(* Logix 5000 project; controller cal1615 1756-L62 rev 20.19; software revision 20.05; part 26 of 82 *)
(* tags used below, declared in another part *)
   AFI : BOOL;   // Always False Bit
   FAULT : BOOL;   // Fault AFI
   p01_param_open_oven_temp : REAL;
   p01_recipe_active : recipe;   // Active Recipe
   p01_sys_enc : SYS_ENC;   // System Encoder
   p01r09_open_oven : BOOL;
   p01r09_pb_global_reset : BOOL;   // System Modes PB: Global Fault Reset
   p01r13_permissive_oxidizer : BOOL;   // System Line Start Sequence Permissive Oxidizer
   p02_dint_from_hmi : hmi_dint;
   p11r30 : routine;   // Zone 1 Temperature Control
   p12_ai_lfl : REAL;   // Zone 2 Analog Input Lower Flash Limit
   p12_ai_tc01 : REAL;   // Zone 2 Analog Input Control Thermocouple 1
   p12_ai_tc02 : REAL;   // Zone 2 Analog Input Control Thermocouple 2
   p12_ao_cv : REAL;   // Zone 2 Analog Output Control Valve
   p12_di_burner_auto : BOOL;   // Zone 2 Digital Input Burner Auto
   p12_di_burner_safeties_ok : BOOL;   // Zone 2 Digital Input Burner Safeties Ok
   p12_di_door_open : BOOL;   // Zone 2 Digital Input Access Door Open
   p12_di_exh : acs800_di_normal;   // Zone 2 Digital Inputs Exhaust Fan
   p12_di_exh_flow_ok : BOOL;   // Zone 2 Digital Input Exhaust Flow OK
   p12_di_flame_failure : BOOL;   // Zone 2 Digital Input Flame Failure
   p12_di_flame_on : BOOL;   // Zone 2 Digital Input Burner is On
   p12_di_high_limit_temp_ok : BOOL;   // Zone 2 Digital Input High Limit Temperature OK
   p12_di_recirc : acs800_di_normal;   // Zone 2 Digital Inputs Recirc Fan
   p12_di_recirc_flow_ok : BOOL;   // Zone 2 Digital Input Recirc Flow OK
   p12_di_sp00 : BOOL;   // Zone 2 Digital Input Combustion Blower Pressure OK
   p12_di_tc01_bo : BOOL;   // Zone 2 Digital Input Control Thermocouple 1 Failure
   p12_di_tc02_bo : BOOL;   // Zone 2 Digital Input Control Thermocouple 2 Failure
   p12_do_enable_burner : BOOL;   // Zone 2 Digital Output Enable Burner
   p12_do_rst_flame : BOOL;   // Zone 2 Digital Output Reset Flame Safety
   p12_param_fast_to_soak : REAL;   // Zone 2 Parameter Fast to Soak Control
   p12_param_lfl_hhl : REAL;   // Zone 2 Parameter High High Lower Flash Limit
   p12_param_pid1_ff : REAL;   // Zone 2 Parameter Fast PID Bias
   p12_param_pid1_kd : REAL;   // Zone 2 Parameter Fast PID Derivative Gain
   p12_param_pid1_ki : REAL;   // Zone 2 Parameter Fast PID Integral Gain
   p12_param_pid1_kp : REAL;   // Zone 2 Parameter Fast PID Proportional Gain
   p12_param_pid2_ff : REAL;   // Zone 2 Parameter Auto PID Bias
   p12_param_pid2_kd : REAL;   // Zone 2 Parameter Auto PID Derivative Gain
   p12_param_pid2_ki : REAL;   // Zone 2 Parameter Auto PID Integral Gain
   p12_param_pid2_kp : REAL;   // Zone 2 Parameter Auto PID Proportional Gain
   p12_param_soak_to_fast : REAL;   // Zone 2 Parameter Soak to Fast Control
   p12_param_tc01_hl : REAL;   // Zone 2 Parameter Process Air High Limit
   p12r01 : routine;   // Zone 2 Main
   p12r02_shutdown_temp : BOOL;   // Zone 2 Misc Control Safe Shutdown Temperature
   p12r10 : routine;   // Zone 2
   p12r10_timer_fault : TIMER[4];   // Zone 2 Fault Delay
   p12r16_pid_temp_cv : DINT;   // Zone 2 Temperature Control Control Valve
   p12r16_temp_ok : BOOL;   // Zone 2 Temperature Control Temperature OK
   p12r20 : routine;   // Zone 2 Temp Sequence
   p12r20_safeties_ok : BOOL;   // Zone 2 Temperature Control Burner Safeties OK this Lightoff
   p12r20_state : DINT;   // Zone 2 Temperature Control State
   p12r20_status : DINT;   // Zone 2 Temperature Control Sequence Status
   p12r20_timer_fault : TIMER[4];   // Zone 2 Temp Sequence Fault Delay
   p12r20_timer_state_11 : TIMER;   // Zone 2 Temp Sequence State 11 Dwell
   p12r20_timer_state_3 : TIMER;   // Zone 2 Temperature Control State 3 Dwell
   p12r20_timer_state_4 : TIMER;   // Zone 2 Temp Sequence State 4 Dwell
   p12r20_timer_state_7 : TIMER;   // Zone 2 Temp Sequence State 7 Dwell
   p12r20_timer_warning : TIMER[4];   // Zone 2 Temp Sequence Warning Delay
   p12r30 : routine;   // Zone 2 Temperature Control
   p12r30_cv_man_sp : REAL;   // Zone 2 Temperature Control Manual Heat Control Valve Setpoint
   p12r30_pb_auto : BOOL;   // Zone 2 Temperature Control PB: Zone Control Auto
   p12r30_pb_manual : BOOL;   // Zone 2 Temperature Control PB: Zone Control Manual
   p12r30_pb_zone_off : BOOL;   // Zone 2 Temperature Control PB: Stop Zone Heat Control
   p12r30_pb_zone_on : BOOL;   // Zone 2 Temperature Control PB: Start Zone Heat Control
   p12r30_permissive_run : BOOL;   // Zone 2 Temperature Control Run Permissive
   p12r30_pid_temp : PID;   // Zone 2 Temperature Control PID
   p12r30_pid_temp_pv : REAL;   // Zone 2 Temperature Control PID Temp Process Variable
   p12r30_pid_temp_sp : REAL;   // Zone 2 Temperature Control PID Temperature Control Setpoint
   p12r30_pid_temp_sp_error : REAL;   // Zone 2 Temperature Control Setpoint/Process Variable Error (ABS)
   p12r30_pid_temp_sp_last : REAL;   // Zone 2 Temperature Control Setpoint Last Scan
   p12r30_request_deviation_warning : BOOL;   // Zone 2 Temperature Control Request Setpoint Deviation Warning
   p12r30_request_heat : BOOL;   // Zone 2 Temperature Control Request Heat
   p12r30_request_heat_last : BOOL;   // Zone 2 Temperature Control Request Heat Last Scan
   p12r30_request_manual : BOOL;   // Zone 2 Temperature Control Request Manual Control
   p12r30_request_PID_shot : BOOL;
   p12r30_request_soak_control : BOOL;   // Zone 2 Temperature Control Request Soak Control
   p12r30_temp_deviation_setpoint : DINT;
   p12r30_timer_fault : TIMER[16];   // Zone 2 Temperature Control Fault Delay
   p12r30_vfds_ok : BOOL;
   p12r31 : routine;   // Zone 2 Exhaust VFD
   p12r32 : routine;   // Zone 2 Recirc VFD
   p23_di_impreg_exhaust_running : BOOL;
   p23_di_impreg_tank_up : BOOL;   // Input Impreg Dip Tank Up
   p23r02 : routine;   // Impreg Misc Control
   p23r13 : routine;
(* P12_Zone_2, continued *)

ROUTINE R20_Temp_Sequence   (* ladder *)
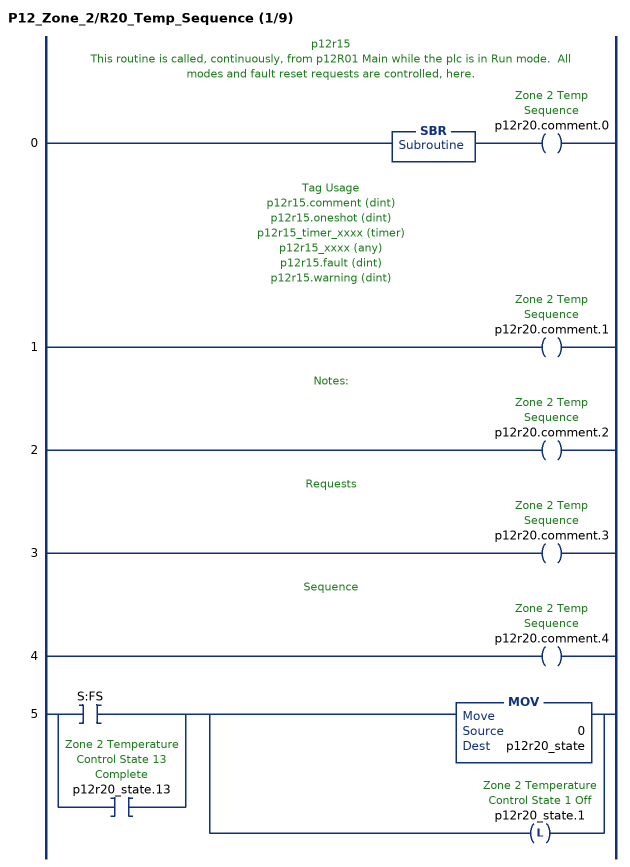
   // p12r15
   // This routine is called, continuously, from p12R01 Main while the plc is in Run mode.  All modes and fault reset requests are controlled, here.
   0: SBR()OTE(p12r20.comment.0);
   // Tag Usage
   // p12r15.comment (dint)
   // p12r15.oneshot (dint)
   // p12r15_timer_xxxx (timer)
   // p12r15_xxxx (any)
   // p12r15.fault (dint)
   // p12r15.warning (dint)
   1: OTE(p12r20.comment.1);
   // Notes:
   2: OTE(p12r20.comment.2);
   // Requests
   3: OTE(p12r20.comment.3);
   // Sequence
   4: OTE(p12r20.comment.4);
   5: [XIC(S:FS) ,XIC(p12r20_state.13) ][MOV(0,p12r20_state) ,OTL(p12r20_state.1) ];
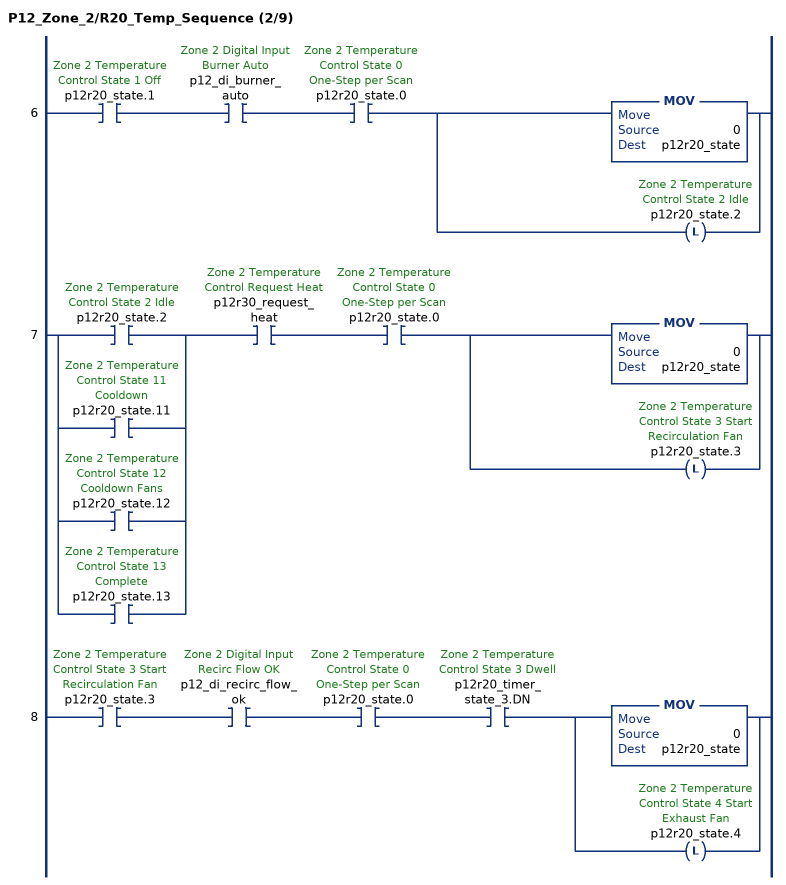
   6: XIC(p12r20_state.1)XIC(p12_di_burner_auto)XIC(p12r20_state.0)[MOV(0,p12r20_state) ,OTL(p12r20_state.2) ];
   7: [XIC(p12r20_state.2) ,XIC(p12r20_state.11) ,XIC(p12r20_state.12) ,XIC(p12r20_state.13) ]XIC(p12r30_request_heat)XIC(p12r20_state.0)[MOV(0,p12r20_state) ,OTL(p12r20_state.3) ];
   8: XIC(p12r20_state.3)XIC(p12_di_recirc_flow_ok)XIC(p12r20_state.0)XIC(p12r20_timer_state_3.DN)[MOV(0,p12r20_state) ,OTL(p12r20_state.4) ];
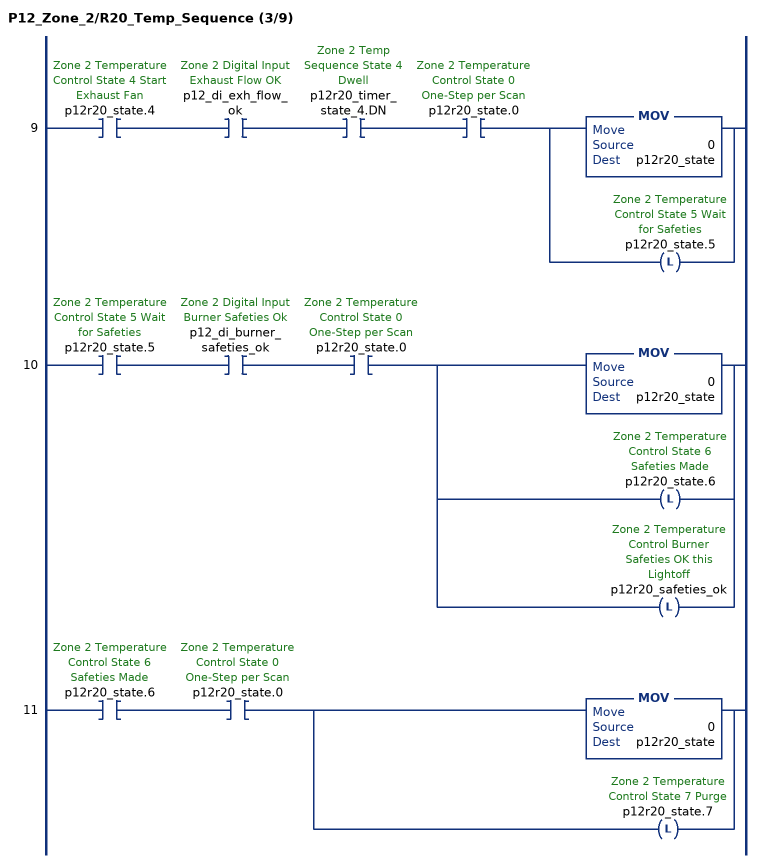
   9: XIC(p12r20_state.4)XIC(p12_di_exh_flow_ok)XIC(p12r20_timer_state_4.DN)XIC(p12r20_state.0)[MOV(0,p12r20_state) ,OTL(p12r20_state.5) ];
   10: XIC(p12r20_state.5)XIC(p12_di_burner_safeties_ok)XIC(p12r20_state.0)[MOV(0,p12r20_state) ,OTL(p12r20_state.6) ,OTL(p12r20_safeties_ok) ];
   11: XIC(p12r20_state.6)XIC(p12r20_state.0)[MOV(0,p12r20_state) ,OTL(p12r20_state.7) ];
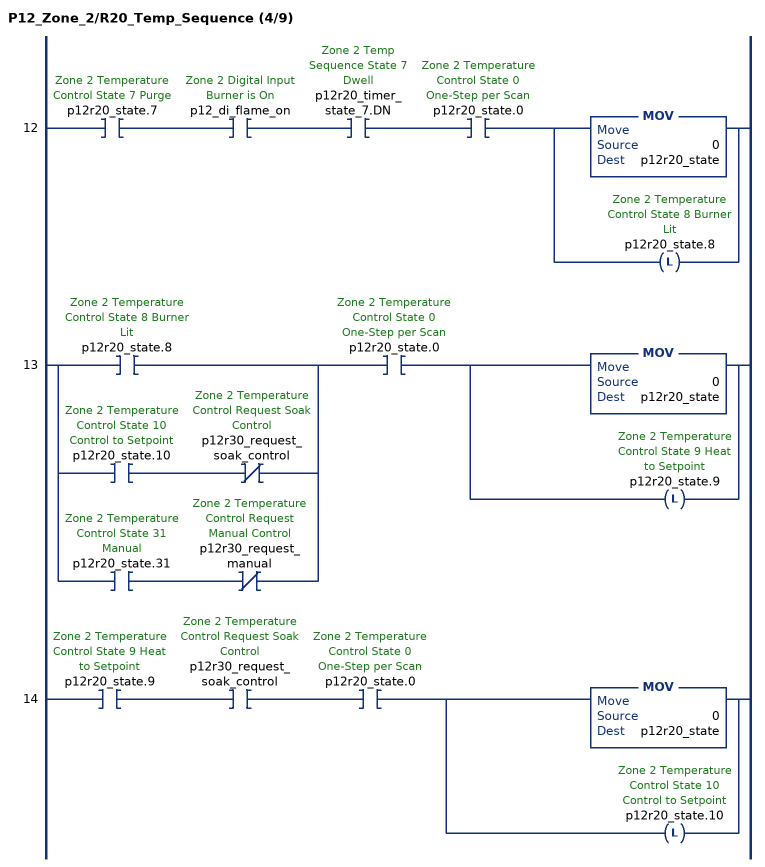
   12: XIC(p12r20_state.7)XIC(p12_di_flame_on)XIC(p12r20_timer_state_7.DN)XIC(p12r20_state.0)[MOV(0,p12r20_state) ,OTL(p12r20_state.8) ];
   13: [XIC(p12r20_state.8) ,XIC(p12r20_state.10) XIO(p12r30_request_soak_control) ,XIC(p12r20_state.31) XIO(p12r30_request_manual) ]XIC(p12r20_state.0)[MOV(0,p12r20_state) ,OTL(p12r20_state.9) ];
   14: XIC(p12r20_state.9)XIC(p12r30_request_soak_control)XIC(p12r20_state.0)[MOV(0,p12r20_state) ,OTL(p12r20_state.10) ];
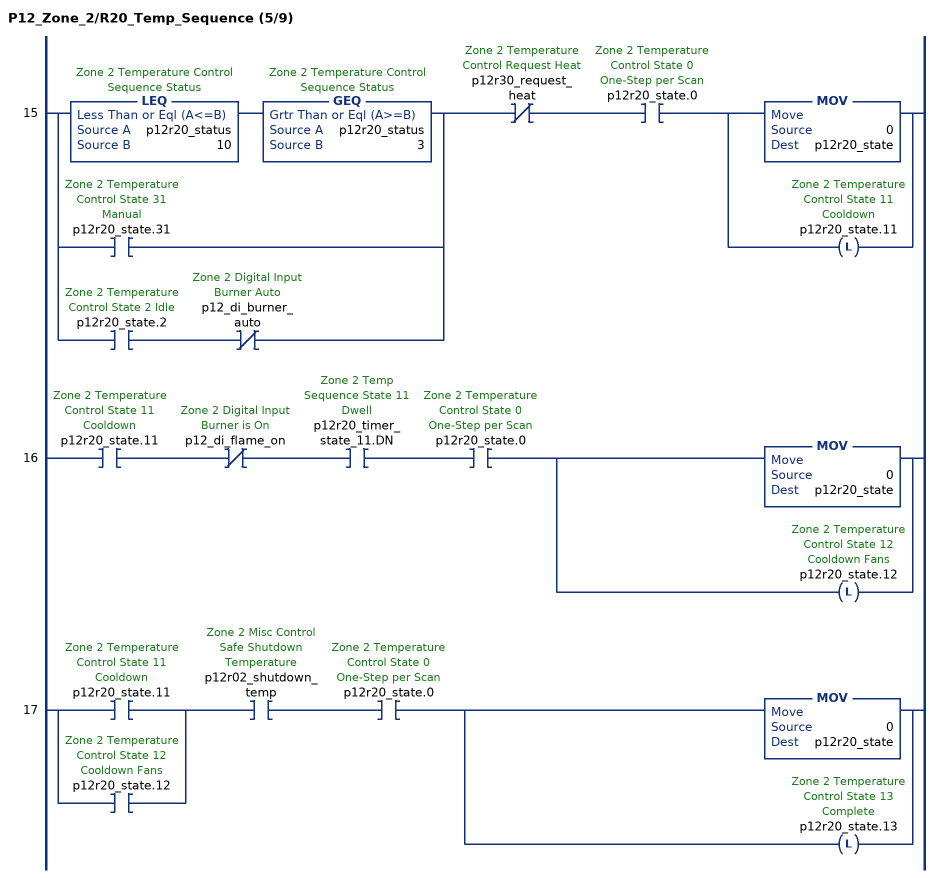
   15: [[LEQ(p12r20_status,10) GEQ(p12r20_status,3) ,XIC(p12r20_state.31) ] ,XIC(p12r20_state.2) XIO(p12_di_burner_auto) ]XIO(p12r30_request_heat)XIC(p12r20_state.0)[MOV(0,p12r20_state) ,OTL(p12r20_state.11) ];
   16: XIC(p12r20_state.11)XIO(p12_di_flame_on)XIC(p12r20_timer_state_11.DN)XIC(p12r20_state.0)[MOV(0,p12r20_state) ,OTL(p12r20_state.12) ];
   17: [XIC(p12r20_state.11) ,XIC(p12r20_state.12) ]XIC(p12r02_shutdown_temp)XIC(p12r20_state.0)[MOV(0,p12r20_state) ,OTL(p12r20_state.13) ];
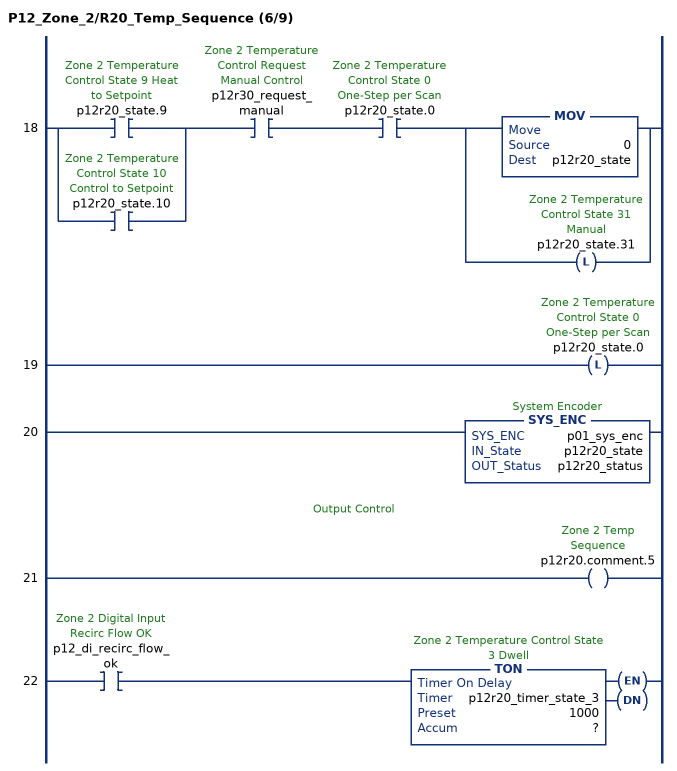
   18: [XIC(p12r20_state.9) ,XIC(p12r20_state.10) ]XIC(p12r30_request_manual)XIC(p12r20_state.0)[MOV(0,p12r20_state) ,OTL(p12r20_state.31) ];
   19: OTL(p12r20_state.0);
   20: SYS_ENC(p01_sys_enc,p12r20_state,p12r20_status);
   // Output Control
   21: OTE(p12r20.comment.5);
   22: XIC(p12_di_recirc_flow_ok)TON(p12r20_timer_state_3,?,?);
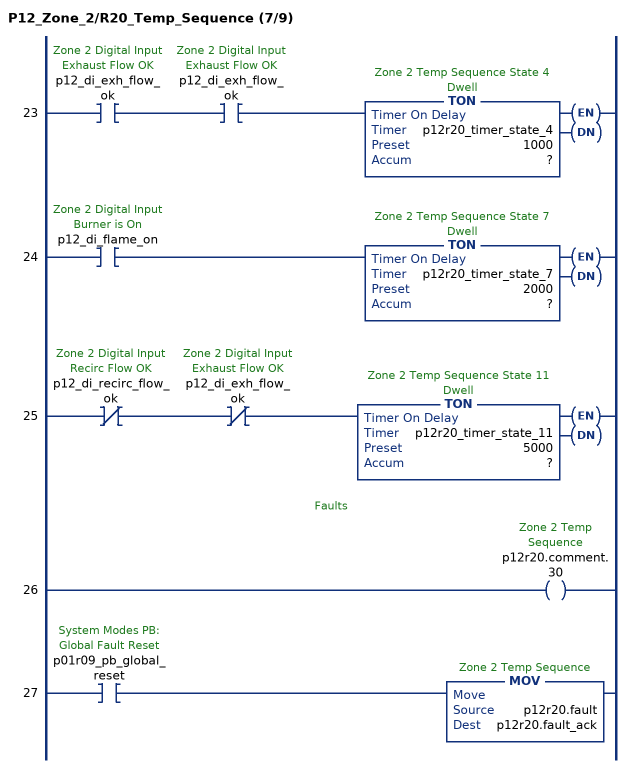
   23: XIC(p12_di_exh_flow_ok)XIC(p12_di_exh_flow_ok)TON(p12r20_timer_state_4,?,?);
   24: XIC(p12_di_flame_on)TON(p12r20_timer_state_7,?,?);
   25: XIO(p12_di_recirc_flow_ok)XIO(p12_di_exh_flow_ok)TON(p12r20_timer_state_11,?,?);
   // Faults
   26: OTE(p12r20.comment.30);
   27: XIC(p01r09_pb_global_reset)MOV(p12r20.fault,p12r20.fault_ack);
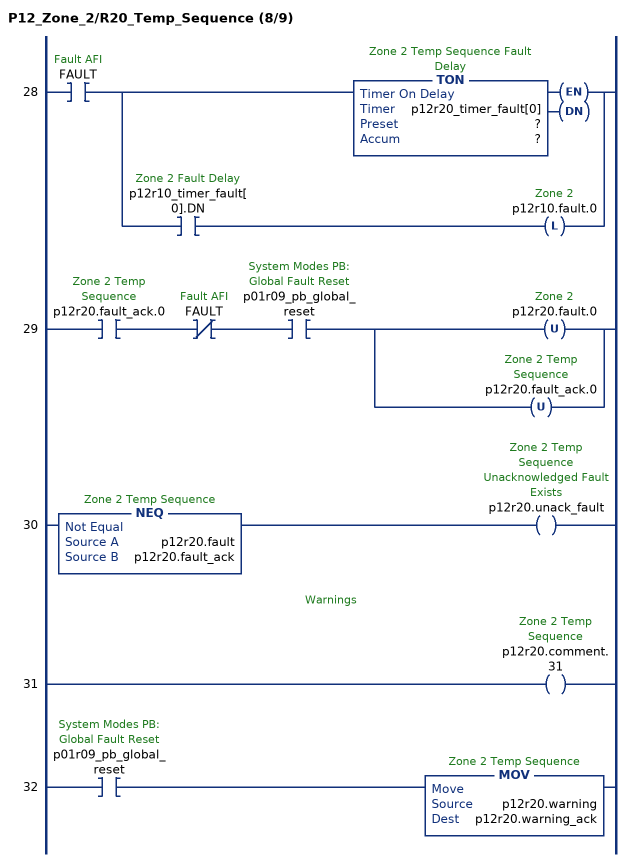
   28: XIC(FAULT)[TON(p12r20_timer_fault[0],?,?) ,XIC(p12r10_timer_fault[0].DN) OTL(p12r10.fault.0) ];
   29: XIC(p12r20.fault_ack.0)XIO(FAULT)XIC(p01r09_pb_global_reset)[OTU(p12r20.fault.0) ,OTU(p12r20.fault_ack.0) ];
   30: NEQ(p12r20.fault,p12r20.fault_ack)OTE(p12r20.unack_fault);
   // Warnings
   31: OTE(p12r20.comment.31);
   32: XIC(p01r09_pb_global_reset)MOV(p12r20.warning,p12r20.warning_ack);
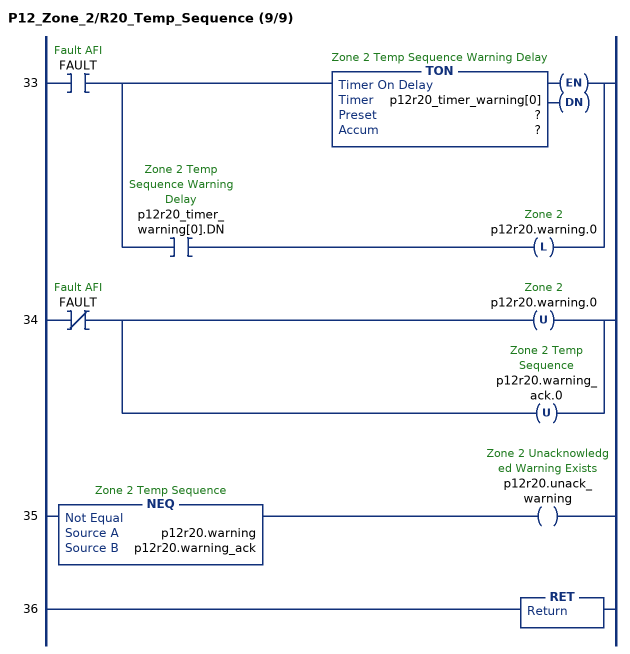
   33: XIC(FAULT)[TON(p12r20_timer_warning[0],?,?) ,XIC(p12r20_timer_warning[0].DN) OTL(p12r20.warning.0) ];
   34: XIO(FAULT)[OTU(p12r20.warning.0) ,OTU(p12r20.warning_ack.0) ];
   35: NEQ(p12r20.warning,p12r20.warning_ack)OTE(p12r20.unack_warning);
   36: RET();
END_ROUTINE

ROUTINE R30_Temperature_Control   (* ladder *)
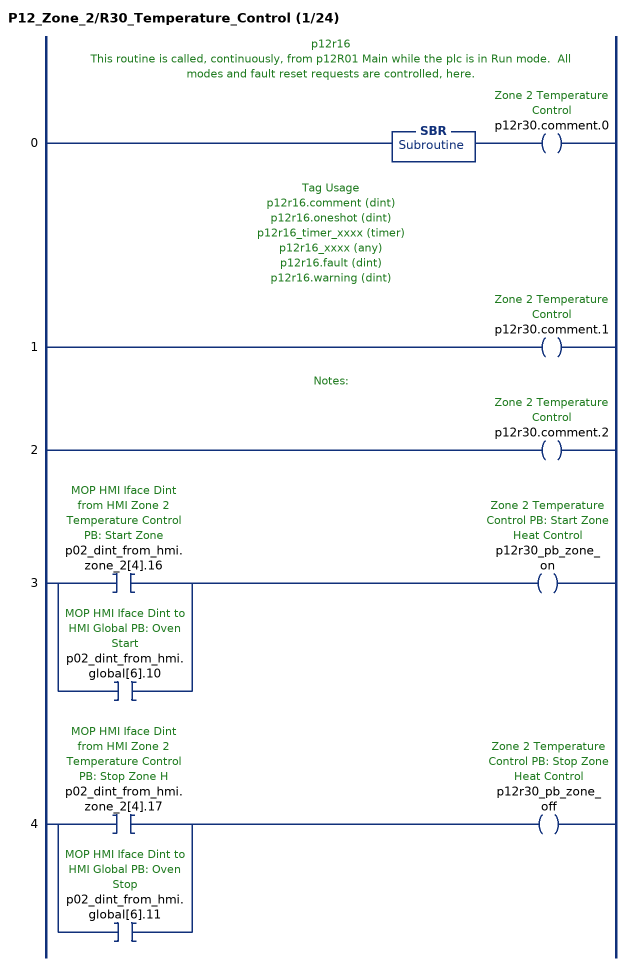
   // p12r16
   // This routine is called, continuously, from p12R01 Main while the plc is in Run mode.  All modes and fault reset requests are controlled, here.
   0: SBR()OTE(p12r30.comment.0);
   // Tag Usage
   // p12r16.comment (dint)
   // p12r16.oneshot (dint)
   // p12r16_timer_xxxx (timer)
   // p12r16_xxxx (any)
   // p12r16.fault (dint)
   // p12r16.warning (dint)
   1: OTE(p12r30.comment.1);
   // Notes:
   2: OTE(p12r30.comment.2);
   3: [XIC(p02_dint_from_hmi.zone_2[4].16) ,XIC(p02_dint_from_hmi.global[6].10) ]OTE(p12r30_pb_zone_on);
   4: [XIC(p02_dint_from_hmi.zone_2[4].17) ,XIC(p02_dint_from_hmi.global[6].11) ]OTE(p12r30_pb_zone_off);
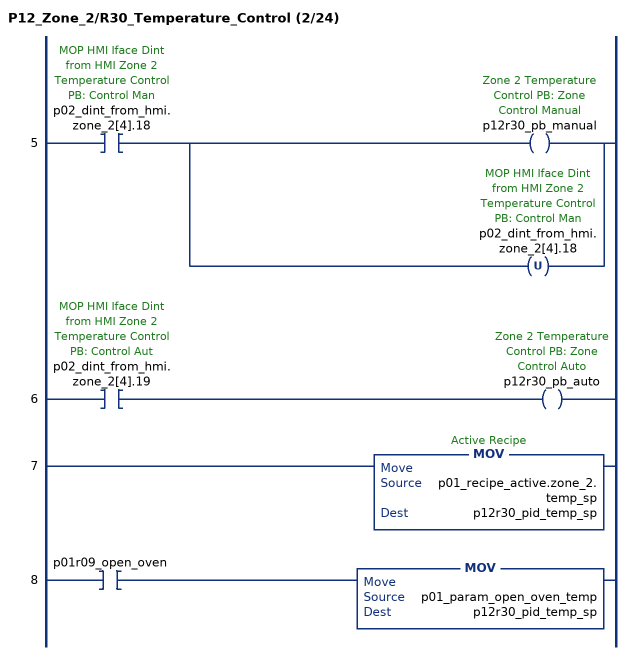
   5: XIC(p02_dint_from_hmi.zone_2[4].18)[OTE(p12r30_pb_manual) ,OTU(p02_dint_from_hmi.zone_2[4].18) ];
   6: XIC(p02_dint_from_hmi.zone_2[4].19)OTE(p12r30_pb_auto);
   7: MOV(p01_recipe_active.zone_2.temp_sp,p12r30_pid_temp_sp);
   8: XIC(p01r09_open_oven)MOV(p01_param_open_oven_temp,p12r30_pid_temp_sp);
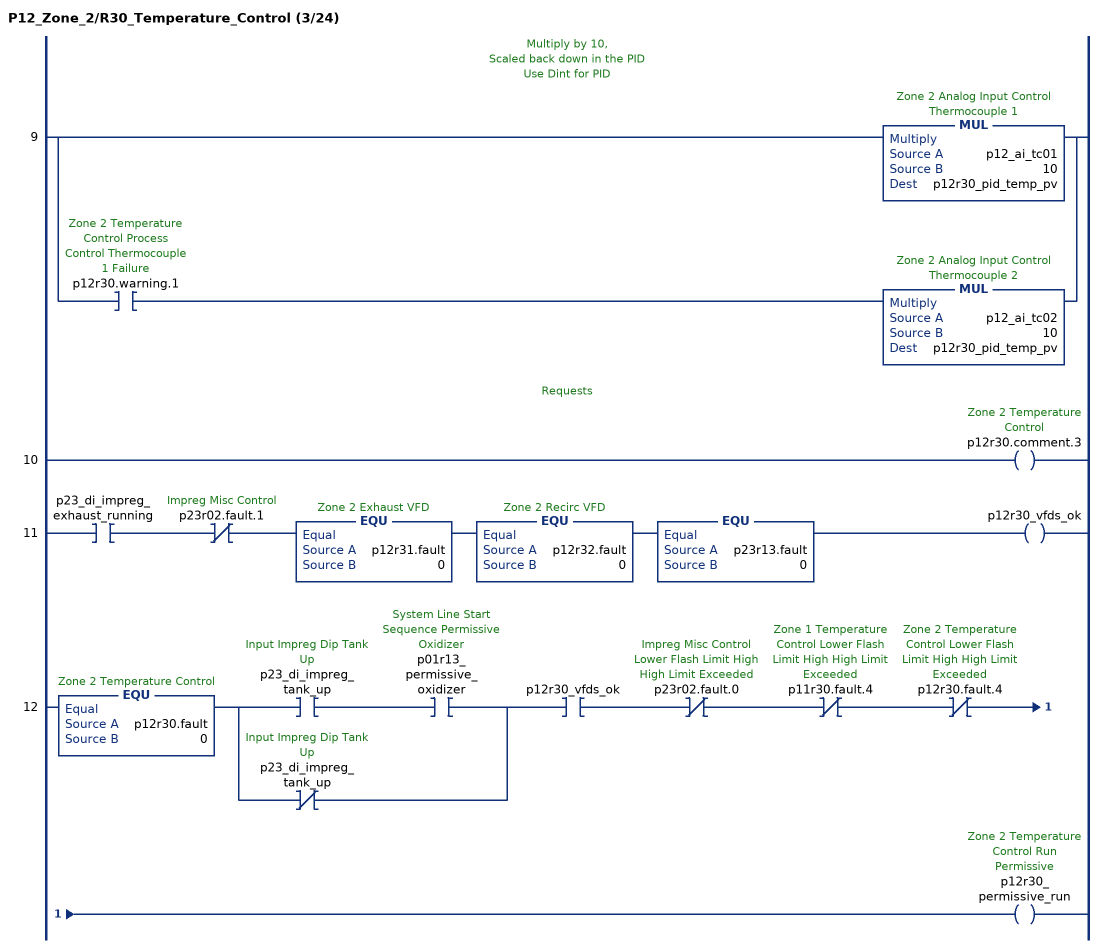
   // Multiply by 10,
   // Scaled back down in the PID
   // Use Dint for PID
   9: [MUL(p12_ai_tc01,10,p12r30_pid_temp_pv) ,XIC(p12r30.warning.1) MUL(p12_ai_tc02,10,p12r30_pid_temp_pv) ];
   // Requests
   10: OTE(p12r30.comment.3);
   11: XIC(p23_di_impreg_exhaust_running)XIO(p23r02.fault.1)EQU(p12r31.fault,0)EQU(p12r32.fault,0)EQU(p23r13.fault,0)OTE(p12r30_vfds_ok);
   12: EQU(p12r30.fault,0)[XIC(p23_di_impreg_tank_up) XIC(p01r13_permissive_oxidizer) ,XIO(p23_di_impreg_tank_up) ]XIC(p12r30_vfds_ok)XIO(p23r02.fault.0)XIO(p11r30.fault.4)XIO(p12r30.fault.4)OTE(p12r30_permissive_run);
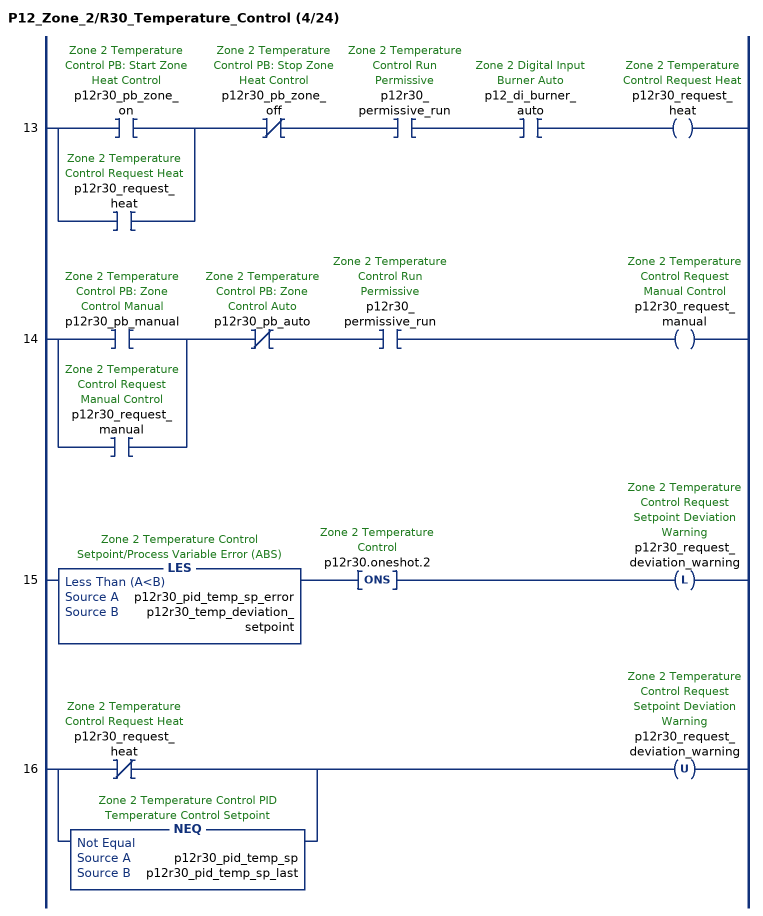
   13: [XIC(p12r30_pb_zone_on) ,XIC(p12r30_request_heat) ]XIO(p12r30_pb_zone_off)XIC(p12r30_permissive_run)XIC(p12_di_burner_auto)OTE(p12r30_request_heat);
   14: [XIC(p12r30_pb_manual) ,XIC(p12r30_request_manual) ]XIO(p12r30_pb_auto)XIC(p12r30_permissive_run)OTE(p12r30_request_manual);
   15: LES(p12r30_pid_temp_sp_error,p12r30_temp_deviation_setpoint)ONS(p12r30.oneshot.2)OTL(p12r30_request_deviation_warning);
   16: [XIO(p12r30_request_heat) ,NEQ(p12r30_pid_temp_sp,p12r30_pid_temp_sp_last) ]OTU(p12r30_request_deviation_warning);
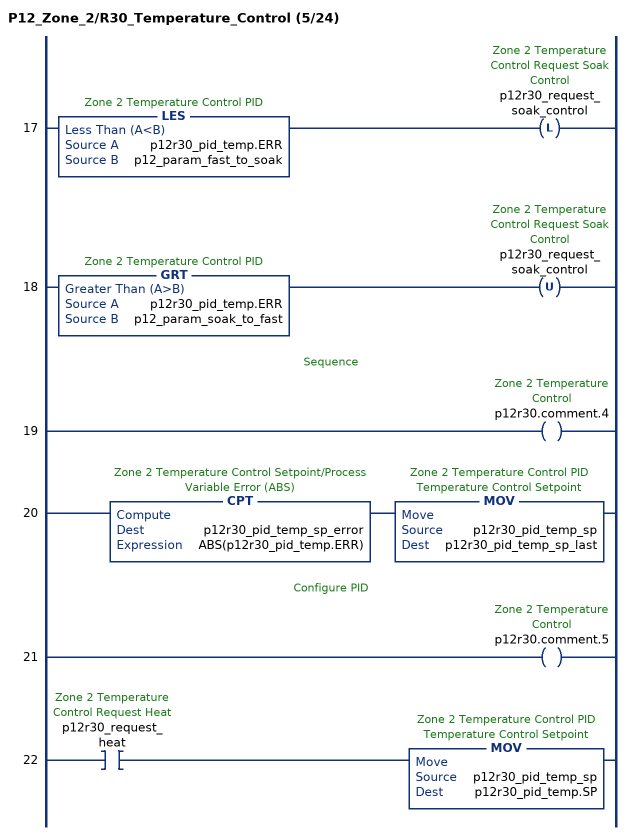
   17: LES(p12r30_pid_temp.ERR,p12_param_fast_to_soak)OTL(p12r30_request_soak_control);
   18: GRT(p12r30_pid_temp.ERR,p12_param_soak_to_fast)OTU(p12r30_request_soak_control);
   // Sequence
   19: OTE(p12r30.comment.4);
   20: CPT(p12r30_pid_temp_sp_error,ABS(p12r30_pid_temp.ERR))MOV(p12r30_pid_temp_sp,p12r30_pid_temp_sp_last);
   // Configure PID
   21: OTE(p12r30.comment.5);
   22: XIC(p12r30_request_heat)MOV(p12r30_pid_temp_sp,p12r30_pid_temp.SP);
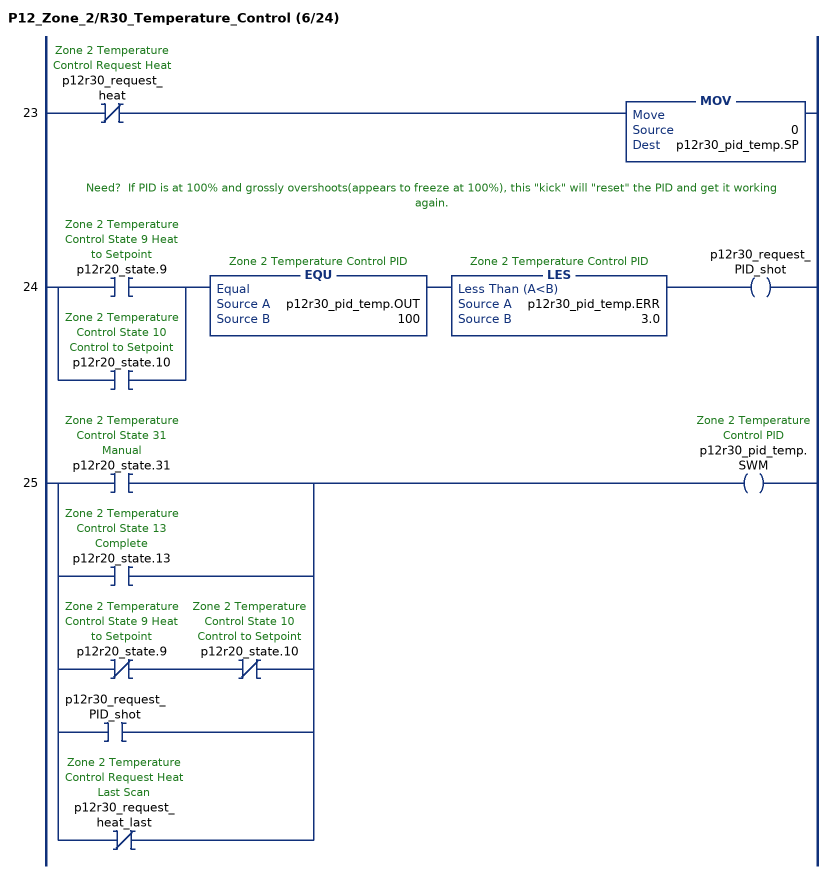
   23: XIO(p12r30_request_heat)MOV(0,p12r30_pid_temp.SP);
   // Need?  If PID is at 100% and grossly overshoots(appears to freeze at 100%), this "kick" will "reset" the PID and get it working again.
   24: [XIC(p12r20_state.9) ,XIC(p12r20_state.10) ]EQU(p12r30_pid_temp.OUT,100)LES(p12r30_pid_temp.ERR,3.0)OTE(p12r30_request_PID_shot);
   25: [XIC(p12r20_state.31) ,XIC(p12r20_state.13) ,XIO(p12r20_state.9) XIO(p12r20_state.10) ,XIC(p12r30_request_PID_shot) ,XIO(p12r30_request_heat_last) ]OTE(p12r30_pid_temp.SWM);
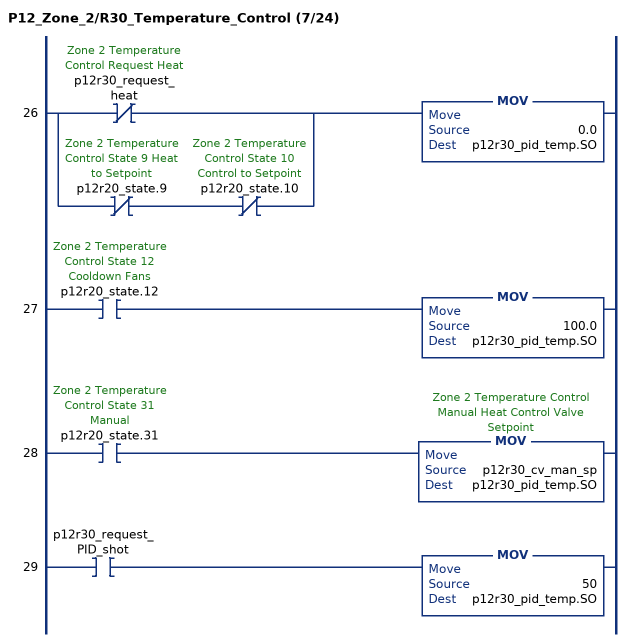
   26: [XIO(p12r30_request_heat) ,XIO(p12r20_state.9) XIO(p12r20_state.10) ]MOV(0.0,p12r30_pid_temp.SO);
   27: XIC(p12r20_state.12)MOV(100.0,p12r30_pid_temp.SO);
   28: XIC(p12r20_state.31)MOV(p12r30_cv_man_sp,p12r30_pid_temp.SO);
   29: XIC(p12r30_request_PID_shot)MOV(50,p12r30_pid_temp.SO);
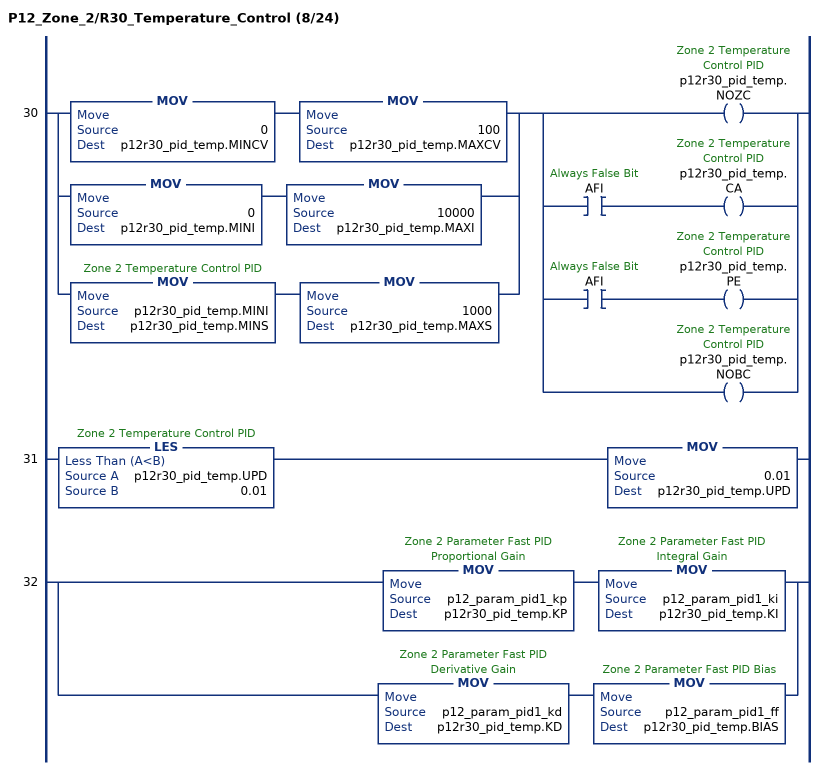
   30: [MOV(0,p12r30_pid_temp.MINCV) MOV(100,p12r30_pid_temp.MAXCV) ,MOV(0,p12r30_pid_temp.MINI) MOV(10000,p12r30_pid_temp.MAXI) ,MOV(p12r30_pid_temp.MINI,p12r30_pid_temp.MINS) MOV(1000,p12r30_pid_temp.MAXS) ][OTE(p12r30_pid_temp.NOZC) ,XIC(AFI) OTE(p12r30_pid_temp.CA) ,XIC(AFI) OTE(p12r30_pid_temp.PE) ,OTE(p12r30_pid_temp.NOBC) ];
   31: LES(p12r30_pid_temp.UPD,0.01)MOV(0.01,p12r30_pid_temp.UPD);
   32: [MOV(p12_param_pid1_kp,p12r30_pid_temp.KP) MOV(p12_param_pid1_ki,p12r30_pid_temp.KI) ,MOV(p12_param_pid1_kd,p12r30_pid_temp.KD) MOV(p12_param_pid1_ff,p12r30_pid_temp.BIAS) ];
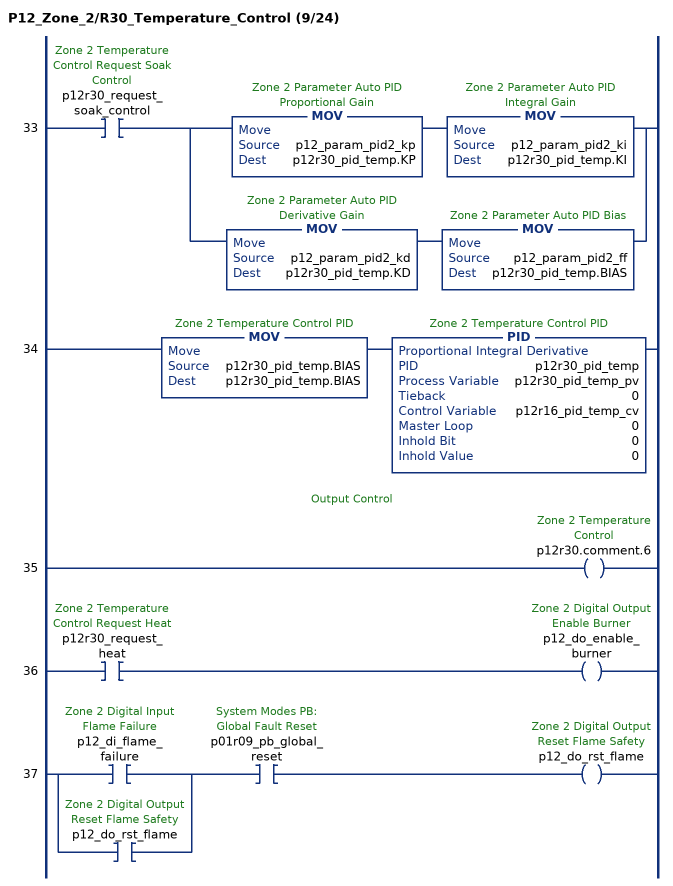
   33: XIC(p12r30_request_soak_control)[MOV(p12_param_pid2_kp,p12r30_pid_temp.KP) MOV(p12_param_pid2_ki,p12r30_pid_temp.KI) ,MOV(p12_param_pid2_kd,p12r30_pid_temp.KD) MOV(p12_param_pid2_ff,p12r30_pid_temp.BIAS) ];
   34: MOV(p12r30_pid_temp.BIAS,p12r30_pid_temp.BIAS)PID(p12r30_pid_temp,p12r30_pid_temp_pv,0,p12r16_pid_temp_cv,0,0,0);
   // Output Control
   35: OTE(p12r30.comment.6);
   36: XIC(p12r30_request_heat)OTE(p12_do_enable_burner);
   37: [XIC(p12_di_flame_failure) ,XIC(p12_do_rst_flame) ]XIC(p01r09_pb_global_reset)OTE(p12_do_rst_flame);
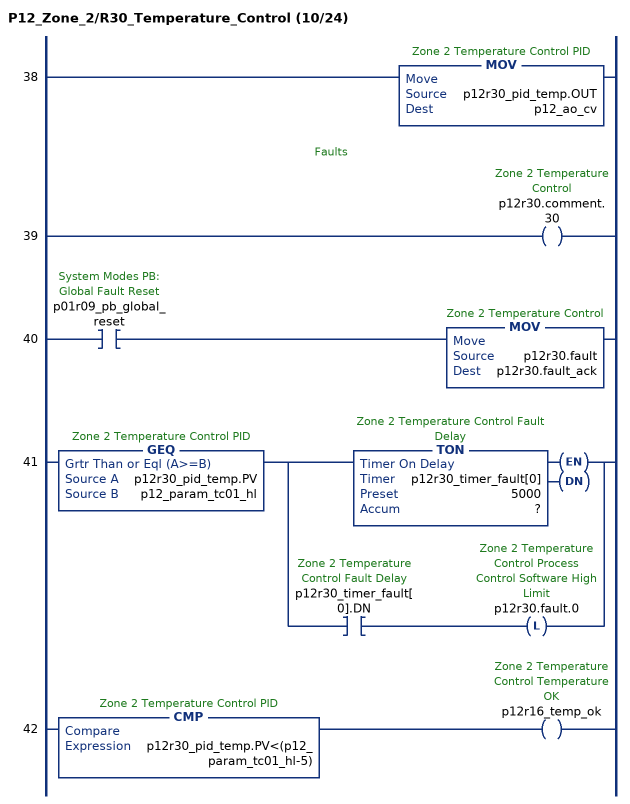
   38: MOV(p12r30_pid_temp.OUT,p12_ao_cv);
   // Faults
   39: OTE(p12r30.comment.30);
   40: XIC(p01r09_pb_global_reset)MOV(p12r30.fault,p12r30.fault_ack);
   41: GEQ(p12r30_pid_temp.PV,p12_param_tc01_hl)[TON(p12r30_timer_fault[0],?,?) ,XIC(p12r30_timer_fault[0].DN) OTL(p12r30.fault.0) ];
   42: CMP(p12r30_pid_temp.PV<(p12_param_tc01_hl-5))OTE(p12r16_temp_ok);
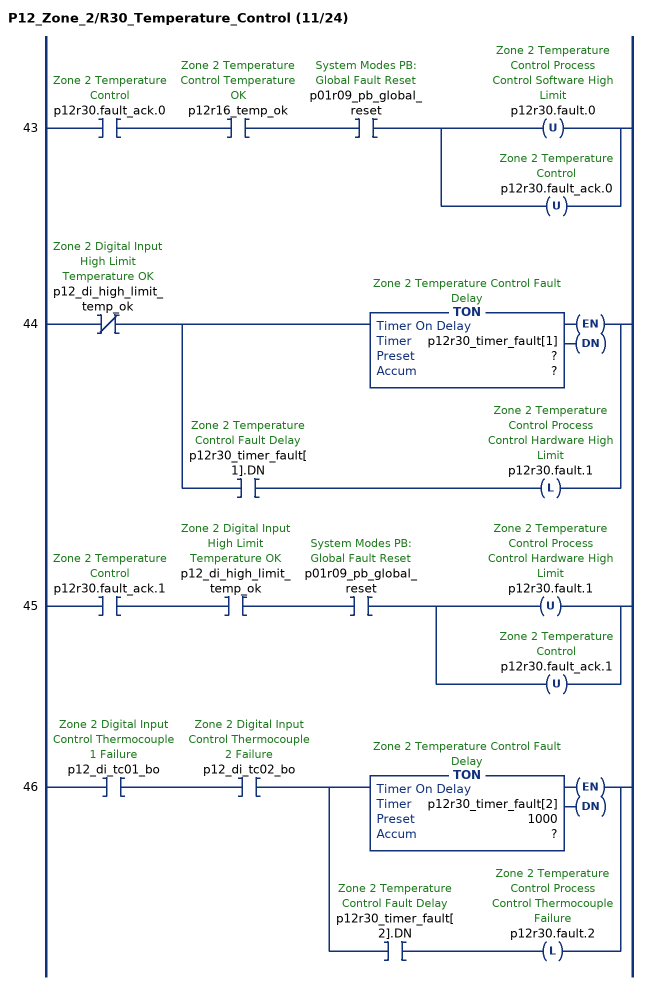
   43: XIC(p12r30.fault_ack.0)XIC(p12r16_temp_ok)XIC(p01r09_pb_global_reset)[OTU(p12r30.fault.0) ,OTU(p12r30.fault_ack.0) ];
   44: XIO(p12_di_high_limit_temp_ok)[TON(p12r30_timer_fault[1],?,?) ,XIC(p12r30_timer_fault[1].DN) OTL(p12r30.fault.1) ];
   45: XIC(p12r30.fault_ack.1)XIC(p12_di_high_limit_temp_ok)XIC(p01r09_pb_global_reset)[OTU(p12r30.fault.1) ,OTU(p12r30.fault_ack.1) ];
   46: XIC(p12_di_tc01_bo)XIC(p12_di_tc02_bo)[TON(p12r30_timer_fault[2],?,?) ,XIC(p12r30_timer_fault[2].DN) OTL(p12r30.fault.2) ];
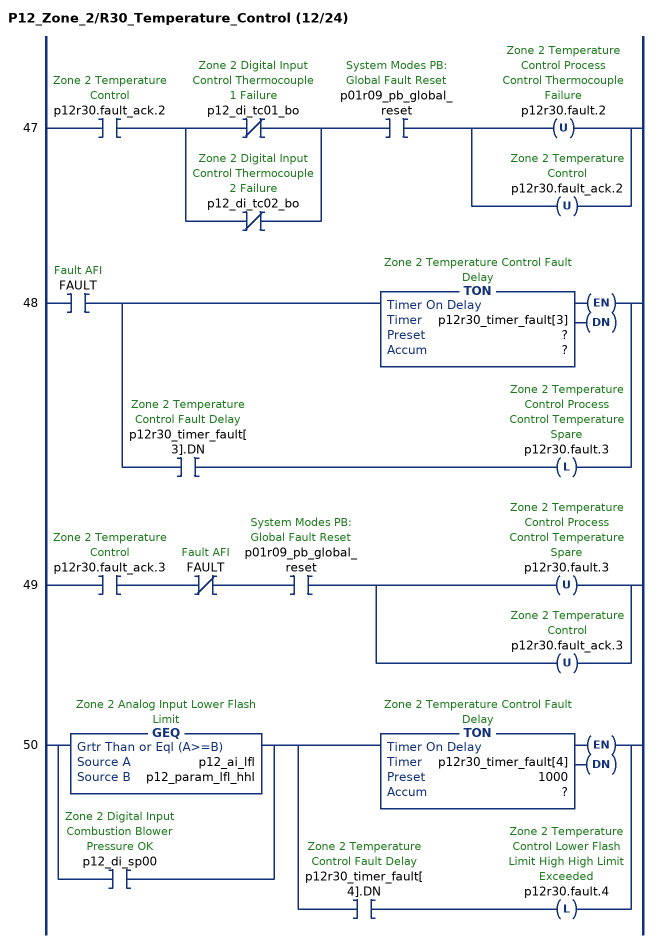
   47: XIC(p12r30.fault_ack.2)[XIO(p12_di_tc01_bo) ,XIO(p12_di_tc02_bo) ]XIC(p01r09_pb_global_reset)[OTU(p12r30.fault.2) ,OTU(p12r30.fault_ack.2) ];
   48: XIC(FAULT)[TON(p12r30_timer_fault[3],?,?) ,XIC(p12r30_timer_fault[3].DN) OTL(p12r30.fault.3) ];
   49: XIC(p12r30.fault_ack.3)XIO(FAULT)XIC(p01r09_pb_global_reset)[OTU(p12r30.fault.3) ,OTU(p12r30.fault_ack.3) ];
   50: [GEQ(p12_ai_lfl,p12_param_lfl_hhl) ,XIC(p12_di_sp00) ][TON(p12r30_timer_fault[4],?,?) ,XIC(p12r30_timer_fault[4].DN) OTL(p12r30.fault.4) ];
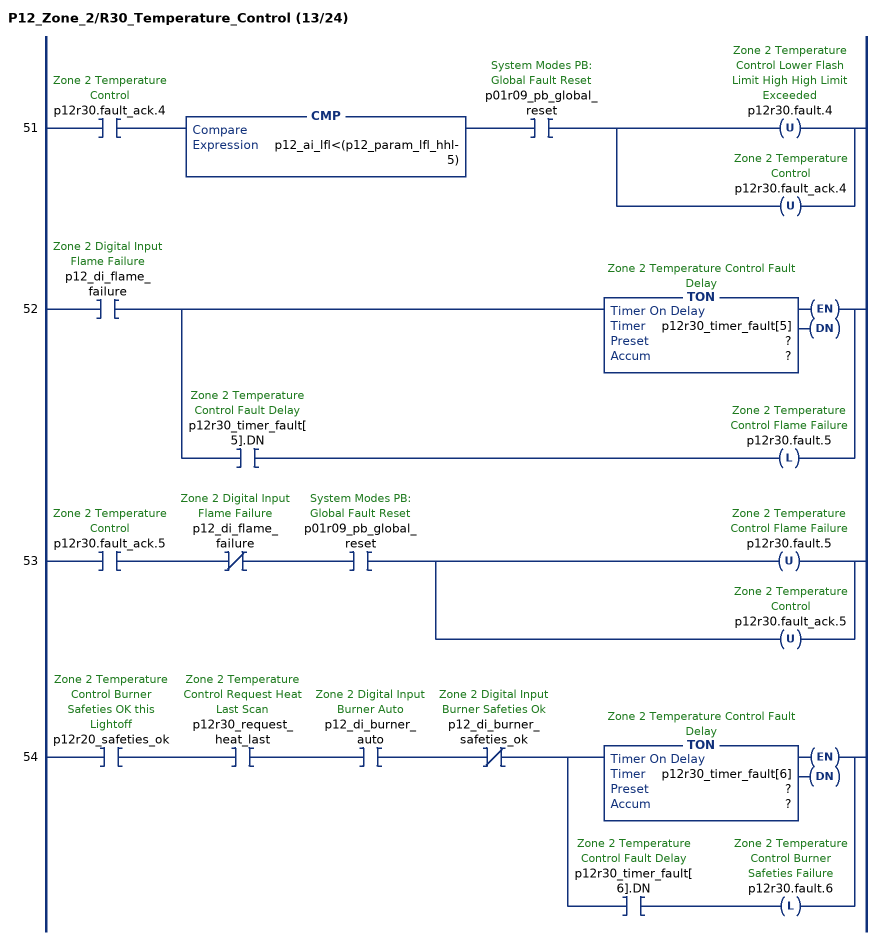
   51: XIC(p12r30.fault_ack.4)CMP(p12_ai_lfl<(p12_param_lfl_hhl-5))XIC(p01r09_pb_global_reset)[OTU(p12r30.fault.4) ,OTU(p12r30.fault_ack.4) ];
   52: XIC(p12_di_flame_failure)[TON(p12r30_timer_fault[5],?,?) ,XIC(p12r30_timer_fault[5].DN) OTL(p12r30.fault.5) ];
   53: XIC(p12r30.fault_ack.5)XIO(p12_di_flame_failure)XIC(p01r09_pb_global_reset)[OTU(p12r30.fault.5) ,OTU(p12r30.fault_ack.5) ];
   54: XIC(p12r20_safeties_ok)XIC(p12r30_request_heat_last)XIC(p12_di_burner_auto)XIO(p12_di_burner_safeties_ok)[TON(p12r30_timer_fault[6],?,?) ,XIC(p12r30_timer_fault[6].DN) OTL(p12r30.fault.6) ];
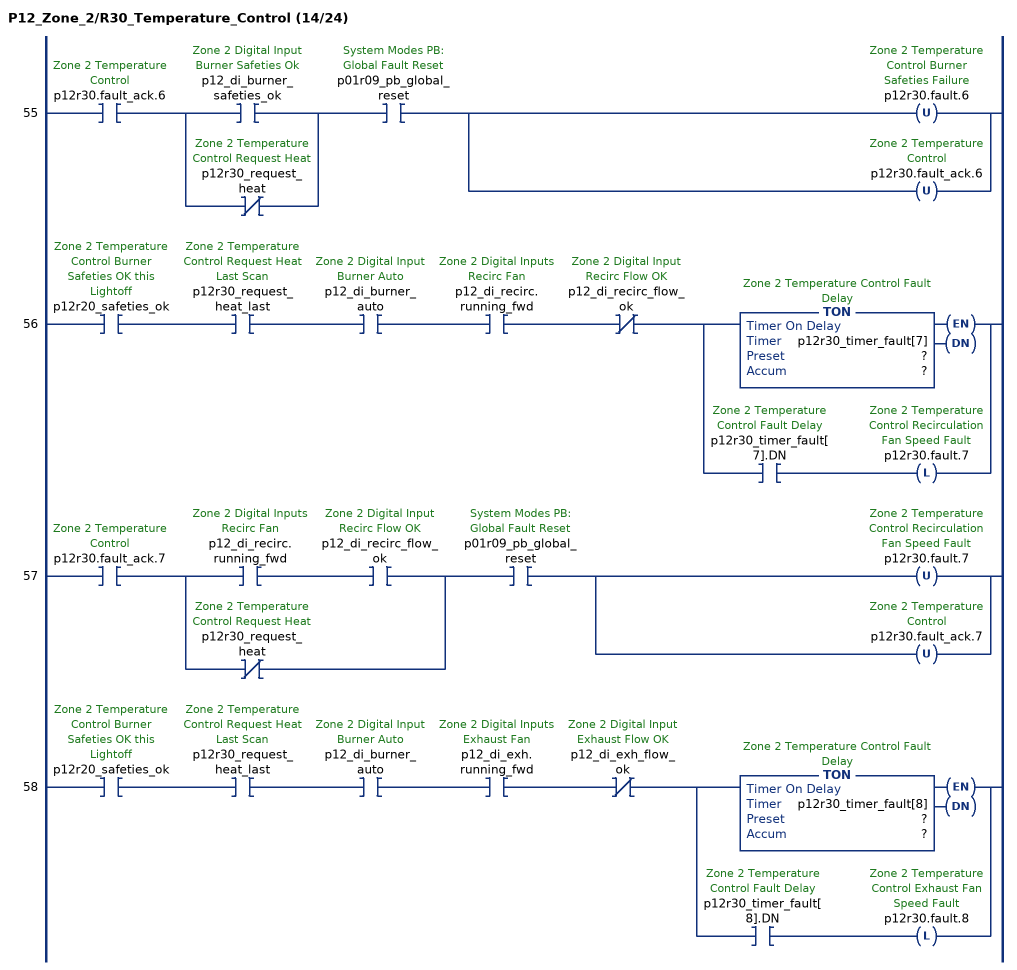
   55: XIC(p12r30.fault_ack.6)[XIC(p12_di_burner_safeties_ok) ,XIO(p12r30_request_heat) ]XIC(p01r09_pb_global_reset)[OTU(p12r30.fault.6) ,OTU(p12r30.fault_ack.6) ];
   56: XIC(p12r20_safeties_ok)XIC(p12r30_request_heat_last)XIC(p12_di_burner_auto)XIC(p12_di_recirc.running_fwd)XIO(p12_di_recirc_flow_ok)[TON(p12r30_timer_fault[7],?,?) ,XIC(p12r30_timer_fault[7].DN) OTL(p12r30.fault.7) ];
   57: XIC(p12r30.fault_ack.7)[XIC(p12_di_recirc.running_fwd) XIC(p12_di_recirc_flow_ok) ,XIO(p12r30_request_heat) ]XIC(p01r09_pb_global_reset)[OTU(p12r30.fault.7) ,OTU(p12r30.fault_ack.7) ];
   58: XIC(p12r20_safeties_ok)XIC(p12r30_request_heat_last)XIC(p12_di_burner_auto)XIC(p12_di_exh.running_fwd)XIO(p12_di_exh_flow_ok)[TON(p12r30_timer_fault[8],?,?) ,XIC(p12r30_timer_fault[8].DN) OTL(p12r30.fault.8) ];
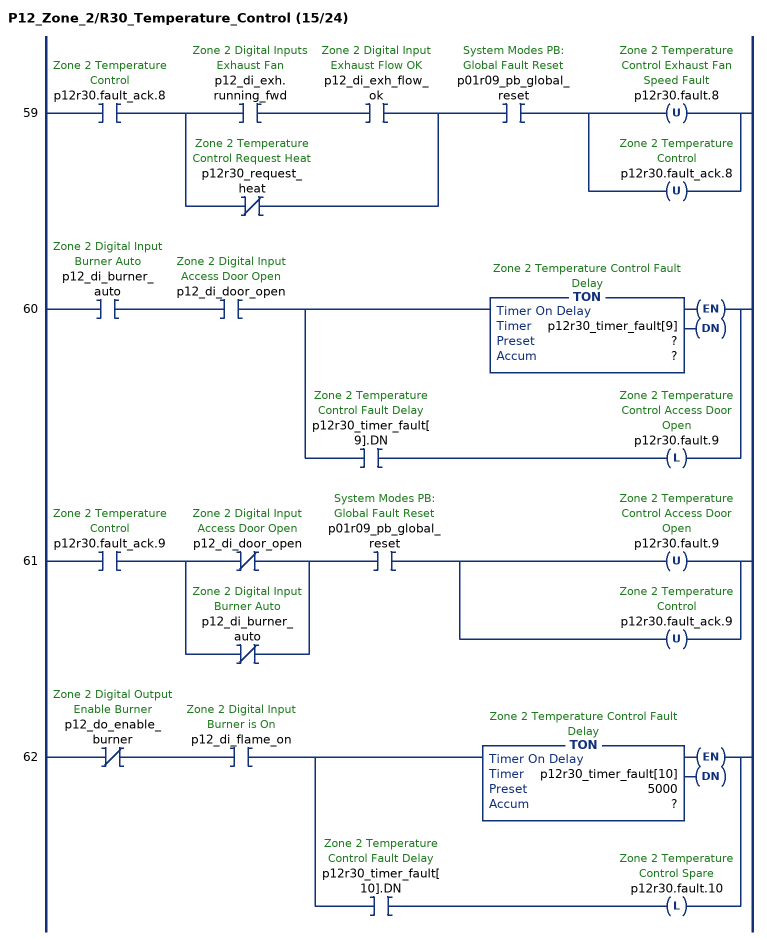
   59: XIC(p12r30.fault_ack.8)[XIC(p12_di_exh.running_fwd) XIC(p12_di_exh_flow_ok) ,XIO(p12r30_request_heat) ]XIC(p01r09_pb_global_reset)[OTU(p12r30.fault.8) ,OTU(p12r30.fault_ack.8) ];
   60: XIC(p12_di_burner_auto)XIC(p12_di_door_open)[TON(p12r30_timer_fault[9],?,?) ,XIC(p12r30_timer_fault[9].DN) OTL(p12r30.fault.9) ];
   61: XIC(p12r30.fault_ack.9)[XIO(p12_di_door_open) ,XIO(p12_di_burner_auto) ]XIC(p01r09_pb_global_reset)[OTU(p12r30.fault.9) ,OTU(p12r30.fault_ack.9) ];
   62: XIO(p12_do_enable_burner)XIC(p12_di_flame_on)[TON(p12r30_timer_fault[10],?,?) ,XIC(p12r30_timer_fault[10].DN) OTL(p12r30.fault.10) ];
